{attribute 'qualified_only'}
{attribute 'strict'}
TYPE E_SafetyState :
(
    INITIALIZING := 0,   // 초기화 중
    NORMAL := 1,         // 정상 상태
    FAULT := 2,          // 고장 상태
    RESETTING := 3       // 리셋 중
) := INITIALIZING;
END_TYPE

(* stored: Version 1.1.0.1
   DUT E_SafetyState: Id {12345678-1234-1234-1234-123456789009} *)
